FUNCTION_BLOCK FB_ProcessCycle
VAR
    eStateInternal      : E_CycleState := E_CycleState.Disabled;

    rtCycleTrigger      : R_TRIG;
    tonSequenceTimeout  : TON;

    bStopPending        			: BOOL;
    bStartIssued        			: BOOL;
    bIndexRequestIssued 			: BOOL;
    bSequenceTimeoutFaultInternal 	: BOOL;

	
END_VAR

METHOD PUBLIC Cyclic
VAR_INPUT
    bEnable                   : BOOL;
    bResetRequest             : BOOL;
    bStopRequest              : BOOL;
    bTwoHandsSafe             : BOOL;
    bSafetyOk                 : BOOL;

    bIndexReady               : BOOL;
    bIndexLocked              : BOOL;
    bIndexBusy                : BOOL;
    bIndexFaulted             : BOOL;
    bStationsIndexPermissive  : BOOL;
    bOperatorIndexPermissive  : BOOL;
    bTemperatureIndexPermissive : BOOL;
    bNestEnableIndexPermissive : BOOL;

    bAllStationsReady         : BOOL;
    bAllStationsComplete      : BOOL;
    bAnyStationFault          : BOOL;
	bHeaterDwellPending 	  : BOOL;

    tSequenceTimeout          : TIME;
END_VAR
VAR_OUTPUT
    bStartStations            : BOOL;
    bStopStations             : BOOL;
    bRequestIndex             : BOOL;

    bCycleActive              : BOOL;
    bCompletePulse            : BOOL;
    bFault                    : BOOL;
    bSequenceTimeoutFault     : BOOL;
    bStopPendingStatus        : BOOL;
    bAutomaticStopRequest     : BOOL;
    bDisabledNestIndexAttempt : BOOL;

    eState                    : E_CycleState;
END_VAR

// Generic indexed-machine process coordinator.
//
// Commissioning sequence aligned with the validated Silicone Station pattern:
//
//   AutoCycle enabled
//      -> initialise
//      -> wait until stations are Ready and supports are physically down
//      -> wait for a FRESH validated two-hand actuation
//      -> validate index permissives
//      -> request ONE index movement
//      -> wait for index complete
//      -> start Patch Dispense / Heat Stake / Vision in parallel
//      -> each station extends its own support
//      -> 3 s simulated process
//      -> each station retracts its support
//      -> all stations Complete
//      -> CycleComplete
//      -> wait for next two-hand actuation
//
// The index FB itself remains the final authority for movement:
// it requires Safety Motion Permitted, Two-Hand Safe, and all station
// supports physically retracted before energising the index outputs.

bStartStations := FALSE;
bStopStations := FALSE;
bRequestIndex := FALSE;
bCompletePulse := FALSE;
bAutomaticStopRequest := FALSE;
bDisabledNestIndexAttempt := FALSE;

rtCycleTrigger(CLK := bTwoHandsSafe);

// ---------------------------------------------------------
// ENABLE / RESET / STOP HANDLING
// ---------------------------------------------------------

IF bResetRequest THEN
    bStopPending := FALSE;
    bStartIssued := FALSE;
    bIndexRequestIssued := FALSE;
    bSequenceTimeoutFaultInternal := FALSE;

    IF bEnable THEN
        eStateInternal := E_CycleState.Initialising;
    ELSE
        eStateInternal := E_CycleState.Disabled;
    END_IF

ELSIF NOT bEnable THEN
    bStopPending := FALSE;
    bStartIssued := FALSE;
    bIndexRequestIssued := FALSE;
    bSequenceTimeoutFaultInternal := FALSE;
    eStateInternal := E_CycleState.Disabled;

ELSE
    // Enter the ProcessCycle automatically when the machine enters AutoCycle.
    IF eStateInternal = E_CycleState.Disabled THEN
        bStopPending := FALSE;
        bStartIssued := FALSE;
        bIndexRequestIssued := FALSE;
        eStateInternal := E_CycleState.Initialising;
    END_IF

    IF bStopRequest THEN
        bStopPending := TRUE;
    END_IF
END_IF

// ---------------------------------------------------------
// FAULT SUPERVISION
// ---------------------------------------------------------

IF bIndexFaulted
    OR bAnyStationFault
    OR (bEnable AND NOT bSafetyOk)
THEN
    eStateInternal := E_CycleState.Fault;
END_IF

// Automatic process-cycle timeout.
//
// This timeout represents OPERATOR INACTIVITY only. It must not run while the
// machine is heating, initialising, indexing, processing, stopping or faulted.
//
// It starts only when the machine is fully ready for the next cycle:
//   - AutoCycle/process coordinator enabled;
//   - waiting for a fresh two-hand operator trigger;
//   - Heat Stake temperature permissive is TRUE;
//   - all process stations are Ready;
//   - index is ready/locked and stationary;
//   - station/index permissives are valid.
//
// Therefore the Heat Stake warm-up time is never included in this timeout.
tonSequenceTimeout(
    IN := bEnable
        AND (eStateInternal = E_CycleState.WaitingForProcessCycleTrigger)
        AND bTemperatureIndexPermissive
        AND bAllStationsReady
        AND bSafetyOk
        AND bIndexReady
        AND bIndexLocked
        AND NOT bIndexBusy
        AND bStationsIndexPermissive
        AND bOperatorIndexPermissive,
    PT := tSequenceTimeout
);

IF tonSequenceTimeout.Q THEN
    // Two minutes of a fully-ready machine waiting for operator activity is
    // NOT a machine fault. Convert it into the same controlled Stop Request
    // philosophy used by the physical Stop button.
    bStopPending := TRUE;
    bAutomaticStopRequest := TRUE;
END_IF

// ---------------------------------------------------------
// PROCESS CYCLE
// ---------------------------------------------------------

CASE eStateInternal OF

    E_CycleState.Disabled:
        // Waiting for machine AutoCycle.

    E_CycleState.Initialising:
        bStartIssued := FALSE;
        bIndexRequestIssued := FALSE;

        // Match the Silicone philosophy:
        // do not arm the operator trigger until the index is stable AND all
        // process tooling is physically in the safe/retracted position.
        IF bSafetyOk
            AND bIndexReady
            AND bIndexLocked
            AND bStationsIndexPermissive
            AND bOperatorIndexPermissive
            AND bTemperatureIndexPermissive
            AND bAllStationsReady
        THEN
            eStateInternal := E_CycleState.WaitingForProcessCycleTrigger;
        END_IF

	E_CycleState.WaitingForProcessCycleTrigger:
	
		IF bStopPending THEN
			eStateInternal := E_CycleState.ControlledStop;
	
		ELSIF bHeaterDwellPending THEN
			// Block new cycles while waiting for Heater Dwell.
			// The machine controller will perform the safe
			// transition to Dwell.

        // The disabled-nest interlock is reported only after a fresh operator
        // index attempt. The machine stays in this state and does not index.
        ELSIF rtCycleTrigger.Q AND NOT bNestEnableIndexPermissive THEN
            bDisabledNestIndexAttempt := TRUE;

        // Fresh two-hand actuation starts the cycle, exactly as on Silicone.
        ELSIF rtCycleTrigger.Q
            AND bSafetyOk
            AND bIndexReady
            AND bIndexLocked
            AND NOT bIndexBusy
            AND bStationsIndexPermissive
            AND bOperatorIndexPermissive
            AND bAllStationsReady
            AND bNestEnableIndexPermissive
        THEN
            eStateInternal := E_CycleState.ValidatingIndexPermissives;
        END_IF

    E_CycleState.ValidatingIndexPermissives:

        IF bStopPending THEN
            eStateInternal := E_CycleState.ControlledStop;
			
		ELSIF bHeaterDwellPending THEN
			// No index movement has been requested yet.
			eStateInternal := E_CycleState.WaitingForProcessCycleTrigger;

        ELSIF NOT bOperatorIndexPermissive THEN
            // A load change cancels this attempt; correction alone cannot reuse held hands.
            eStateInternal := E_CycleState.WaitingForProcessCycleTrigger;

        ELSIF bSafetyOk
            AND bStationsIndexPermissive
            AND bOperatorIndexPermissive
            AND bTemperatureIndexPermissive
            AND bNestEnableIndexPermissive
            AND bIndexReady
            AND bIndexLocked
            AND NOT bIndexBusy
        THEN
            eStateInternal := E_CycleState.RequestingIndexMove;
        END_IF

    E_CycleState.RequestingIndexMove:
        IF bStopPending THEN
            eStateInternal := E_CycleState.ControlledStop;
        ELSIF bSafetyOk AND bStationsIndexPermissive AND bOperatorIndexPermissive
            AND bTemperatureIndexPermissive AND bNestEnableIndexPermissive
            AND bIndexReady AND bIndexLocked AND NOT bIndexBusy AND bTwoHandsSafe
            AND NOT bHeaterDwellPending THEN
            bRequestIndex := TRUE;
            bIndexRequestIssued := TRUE;
            eStateInternal := E_CycleState.WaitingForIndexStart;
        ELSE
            // No request is queued with an invalid load or stale two-hand actuation.
            bIndexRequestIssued := FALSE;
            eStateInternal := E_CycleState.WaitingForProcessCycleTrigger;
        END_IF

    E_CycleState.WaitingForIndexStart:

        IF bStopPending THEN
            eStateInternal := E_CycleState.ControlledStop;

        ELSIF bIndexBusy THEN
            eStateInternal := E_CycleState.WaitingForIndexComplete;
        END_IF

    E_CycleState.WaitingForIndexComplete:

        IF bStopPending THEN
            eStateInternal := E_CycleState.ControlledStop;

        ELSIF NOT bIndexBusy
            AND bIndexReady
            AND bIndexLocked
        THEN
            bIndexRequestIssued := FALSE;
            eStateInternal := E_CycleState.PreparingProcessStations;
        END_IF

    E_CycleState.PreparingProcessStations:

        // After the index has locked in its new position, ensure all three
        // station objects are ready before issuing process start.
        IF bStopPending THEN
            eStateInternal := E_CycleState.ControlledStop;

        ELSIF bAllStationsReady THEN
            eStateInternal := E_CycleState.StartingProcesses;
        END_IF

    E_CycleState.StartingProcesses:
        // If Stop was requested before any station actually started, do not
        // launch a new process. Go directly to the controlled-stop path.
        IF bStopPending THEN
            eStateInternal := E_CycleState.ControlledStop;
        ELSE
            bStartStations := TRUE;
            bStartIssued := TRUE;
            eStateInternal := E_CycleState.WaitingForProcessesRunning;
        END_IF

    E_CycleState.WaitingForProcessesRunning:

        // A Stop Request is intentionally only LATCHED while a station is
        // running. Never interrupt an active station process. The process is
        // allowed to reach its normal Complete state and retract its tooling.
        //
        // IMPORTANT:
        // If no physical nest at any process station contains a part, all
        // stations are intentionally skipped. In that case
        // bAllStationsReady remains TRUE forever, while
        // bAllStationsComplete is already TRUE.
        IF bAllStationsComplete THEN
            eStateInternal := E_CycleState.WaitingForProcessesComplete;

        // Normal case: at least one required station has left Ready and
        // entered its process sequence.
        ELSIF NOT bAllStationsReady THEN
            eStateInternal := E_CycleState.WaitingForProcessesComplete;
        END_IF

    E_CycleState.WaitingForProcessesComplete:

        // Even with Stop pending, allow every active station to finish its
        // normal sequence. Only after all stations are Complete and all
        // supports are physically retracted may the stop proceed.
        IF bAllStationsComplete
            AND bStationsIndexPermissive
        THEN
            bStartIssued := FALSE;
            eStateInternal := E_CycleState.CycleComplete;
        END_IF

    E_CycleState.CycleComplete:
        bCompletePulse := TRUE;

        IF bStopPending THEN
            eStateInternal := E_CycleState.ControlledStop;
        ELSE
            eStateInternal := E_CycleState.WaitingForProcessCycleTrigger;
        END_IF

    E_CycleState.ControlledStop:
        bStopStations := TRUE;

        // Safe stop is complete only when the index has stopped and every
        // support cylinder is physically retracted.
        IF NOT bIndexBusy
            AND bStationsIndexPermissive
        THEN
            bStopPending := FALSE;
            eStateInternal := E_CycleState.Disabled;
        END_IF

    E_CycleState.Fault:
        bStopStations := TRUE;

ELSE
    eStateInternal := E_CycleState.Fault;

END_CASE

bCycleActive :=
    (eStateInternal <> E_CycleState.Disabled)
    AND (eStateInternal <> E_CycleState.Fault);

bFault := (eStateInternal = E_CycleState.Fault);
bSequenceTimeoutFault := bSequenceTimeoutFaultInternal;
bStopPendingStatus := bStopPending;
eState := eStateInternal;
END_METHOD

END_FUNCTION_BLOCK

(* stored: Version 1.1.0.1, ProductVersion 3.1.4026.18
   POU FB_ProcessCycle: Id {622f2bef-5510-4430-be8a-312a17e95422}, SpecialFunc None
   Method Cyclic: Id {e84fc6ef-4070-40dd-8010-e10d3773e159} *)
